INTERFACE ITF_BaseComponent

METHOD activate : BOOL
VAR_INPUT
END_VAR
END_METHOD

METHOD cleanup : BOOL
VAR_INPUT
END_VAR
END_METHOD

METHOD configure : BOOL
VAR_INPUT
END_VAR
END_METHOD

METHOD create : BOOL
VAR_INPUT
END_VAR
END_METHOD

METHOD deactivate : BOOL
VAR_INPUT
END_VAR
END_METHOD

METHOD destroy : BOOL
VAR_INPUT
END_VAR
END_METHOD

METHOD ID : UINT
VAR_INPUT
END_VAR
END_METHOD

PROPERTY name : String
GET
END_GET
END_PROPERTY

METHOD onActivate : BOOL
VAR_INPUT
END_VAR
END_METHOD

METHOD onCleanup : BOOL
VAR_INPUT
END_VAR
END_METHOD

METHOD onConfigure : BOOL
VAR_INPUT
END_VAR
END_METHOD

METHOD onDeactivate : BOOL
VAR_INPUT
END_VAR
END_METHOD

METHOD onError : BOOL
VAR_INPUT
END_VAR
END_METHOD

METHOD onShutdown : BOOL
VAR_INPUT
END_VAR
END_METHOD

PROPERTY path : String
GET
END_GET
END_PROPERTY

METHOD shutdown : BOOL
VAR_INPUT
END_VAR
END_METHOD

PROPERTY state : eState
GET
END_GET
END_PROPERTY

END_INTERFACE

(* stored: Version 1.1.0.1, ProductVersion 3.1.4026.18
   Itf ITF_BaseComponent: Id {65885d39-4024-4344-a8ab-374a6ccc4c59}
   Folder Activities: Id {5e3aa71c-ec0e-47b3-8f33-f08f0fb99381}
   Folder Transitions: Id {6560e606-0171-480a-9918-20910c0e5bdf}
   Method activate: Id {421c2108-8179-4a12-ba41-35989c996212}
   Method cleanup: Id {2b58a7de-95d9-467c-85d1-db9dec921482}
   Method configure: Id {e50a6f49-0903-48ba-8271-1c9d1e1e510c}
   Method create: Id {f7eeaace-e47d-40b3-b2a6-4bfd02509cfb}
   Method deactivate: Id {543d663f-3433-4738-bb10-46e710584fb3}
   Method destroy: Id {8dc262df-163a-4e11-9777-3fbb1a531627}
   Method ID: Id {d32cf108-e71a-41f2-b199-e347f32e6fca}
   Property name: Id {8e02e470-71da-44a6-a68f-092954d86151}
   Get Get: Id {7f1ff7dd-a478-4f29-885d-9677ae5d4a7e}
   Method onActivate: Id {db5ccdf9-dda4-4656-8a40-44601294dbda}
   Method onCleanup: Id {aeb6ee92-c260-499d-8c85-ecf0511ec7d2}
   Method onConfigure: Id {5400f4d2-21c5-44f4-af11-064140524d3d}
   Method onDeactivate: Id {f1a21cdc-6225-4962-9570-04e28e96710c}
   Method onError: Id {6370aa46-a510-420e-b2b1-4a92b9216869}
   Method onShutdown: Id {6b29e55c-0bb5-4ed2-8d4c-29a2f4547848}
   Property path: Id {755b1bdf-ea5e-45d8-b845-25d127de2ac2}
   Get Get: Id {bdac12b3-22bb-41f6-8039-bf0761521d8e}
   Method shutdown: Id {d44b7757-327e-4329-96cc-8c180a9fb4f3}
   Property state: Id {4c5eddbd-3571-4017-85b4-cee88242beba}
   Get Get: Id {42aa47ea-f1d7-4040-ade8-b3efc7baaa84} *)
